(* CODESYS project e!C_Trace_Test_1.ECP

Project tree, tasks and I/O mapping:
  PFC200_CS_2ETH_RS_CAN_DPS : 750-8206 PFC200 2ETH RS CAN DPS, WAGO, order no. 0750-8206, version 5.11.1.16
    application Application
      libraries: ; VisuDialogs, * (System)
      task PLC_Task (cyclic, interval t#10ms, priority 13) calls PLC_PRG
      task VISU_TASK (cyclic, interval T#100ms, priority 15) calls VISU_PRG
      task TRACE_TASK (cyclic, interval T#50ms, priority 14) calls TraceTask
      program PLC_PRG [ST]
      visualisation VisuTrace
      program TraceTest [ST]
      visualisation VisuMix
      program TraceTask [ST]
    DeviceAdapter
    Kbus : Kbus, WAGO, version 1.4.0.2
        unmapped channels: K-BUS diagnostics
      _8_DO_DI_Generic : 075x-8DO8DI, WAGO, order no. 075x-8DO8DI, version 0.0.0.13
          settings: K-BUS Module slot index = 1
          unmapped channels: _IN, _OUT
        DeviceAdapter
      _4_AO_0_10V_DC : 0750-0559, WAGO, order no. 0750-0559, version 0.0.0.13
          settings: K-BUS Module slot index = 2
          unmapped channels: _QW 1, _QW 2, _QW 3, _QW 4
        DeviceAdapter
      _4_AI_10V_DC_s_e : 0750-0457, WAGO, order no. 0750-0457, version 0.0.0.9
          settings: K-BUS Module slot index = 3
          unmapped channels: _IW 1, _IW 2, _IW 3, _IW 4
        DeviceAdapter
      RS_232_RS_485_Interface_adjustable : 0750-0652, WAGO, order no. 0750-0652, version 0.0.0.25
          settings: K-BUS Module slot index = 4
          unmapped channels: _INPUTCHANNEL, _OUTPUTCHANNEL
        DeviceAdapter
    MODBUS
      MODBUS : MODBUS, WAGO, order no. n/a, version 1.1.1.15
    PROFIBUS
      PROFIBUS : PROFIBUS, WAGO, version 1.0.0.0 (disabled)
    CANbus
    Serial
      COM1 : COM1, WAGO, version 0.0.0.19
  libraries: WagoVisuIcons, 1.0.0.8 (WAGO)
  text list GlobalTextList
*)

// PFC200_CS_2ETH_RS_CAN_DPS/Application/PLC_PRG
PROGRAM PLC_PRG
VAR

	xShowUrl: BOOL;
	sUrl: STRING := 'http://192.168.1.32/plc/webvisu.htm';

END_VAR




sUrl;
xShowUrl;

END_PROGRAM

// PFC200_CS_2ETH_RS_CAN_DPS/Application/TraceTask
PROGRAM TraceTask
VAR
END_VAR



TraceTest();
;

END_PROGRAM

// PFC200_CS_2ETH_RS_CAN_DPS/Application/TraceTest
PROGRAM TraceTest
VAR
	rAngle: REAL;
	rSine: REAL;
	TON_SineSample: TON;
	tSineSample: TIME := T#200MS;
	xTraceRecord: BOOL;
END_VAR



xTraceRecord;

TON_SineSample(IN:= TRUE, PT:= tSineSample);
IF (TON_SineSample.Q = TRUE) THEN
	TON_SineSample(IN:= FALSE);
	rAngle := rAngle + 0.1;
END_IF

rSine := 10 * SIN(rAngle);

END_PROGRAM

// PFC200_CS_2ETH_RS_CAN_DPS/Application/VisuTrace
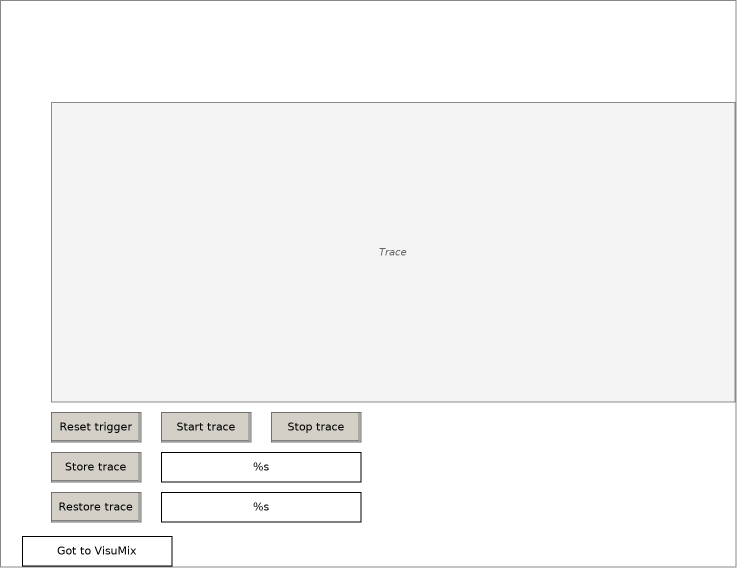
VISUALIZATION VisuTrace  // 737x568
VAR_IN_OUT
END_VAR
VAR
	bResetTrigger : BOOL;
	bStart : BOOL;
	bStop : BOOL;
	bStore : BOOL;
	sStoreFilename : STRING;
	bRestore : BOOL;
	sRestoreFilename : STRING;
END_VAR
    RoundedRectangle (22,536 150x30), "Got to VisuMix"
        OnMouseDown:  Assign=VisuMix, Type=Assignment
    Trace (51,102 684x300)
        p3825648158: bResetTrigger
        p866368322: bStart
        p3851742229: bStop
        p2132035699: bStore
        p163910951: sStoreFilename
        p2217859334: bRestore
        p1301606187: sRestoreFilename
    Button (51,412 90x30), "Reset trigger"
        toggle bResetTrigger
    Button (161,412 90x30), "Start trace"
        toggle bStart
        OnMouseDown: execute { TraceTest.xTraceRecord := TRUE; }
    Button (271,412 90x30), "Stop trace"
        toggle bStop
        OnMouseDown: execute { TraceTest.xTraceRecord := FALSE; }
    Button (51,452 90x30), "Store trace"
        toggle bStore
    Rectangle (161,452 200x30), "%s", text variable: sStoreFilename
        OnMouseClick: write the text variable via Edit
    Button (51,492 90x30), "Restore trace"
        toggle bRestore
    Rectangle (161,492 200x30), "%s", text variable: sRestoreFilename
        OnMouseClick: write the text variable via Edit
END_VISUALIZATION

// PFC200_CS_2ETH_RS_CAN_DPS/Application/VisuMix
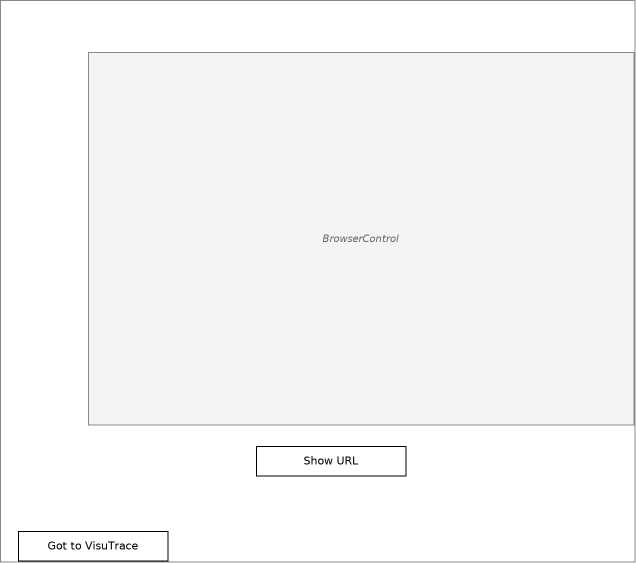
VISUALIZATION VisuMix  // 636x563
    RoundedRectangle (18,531 150x30), "Got to VisuTrace"
        OnMouseDown:  Assign=VisuTrace, Type=Assignment
    BrowserControl (88,52 546x373)
        p3734058945: PLC_PRG.sUrl
        p2179181546: PLC_PRG.xShowUrl
    RoundedRectangle (256,446 150x30), "Show URL"
        toggle PLC_PRG.xShowUrl
END_VISUALIZATION
